{attribute 'qualified_only'}
{attribute 'strict'}
TYPE E_NoveltyDetectorType :
(
	KMPP := 0,
	KNN,
	LBG,
	NBC,
	STA,
	SVM
);
END_TYPE

(* stored: Version 1.1.0.1, ProductVersion 3.1.4024.12
   DUT E_NoveltyDetectorType: Id {b52dccab-d2ed-4c5e-9dae-8b721c3cc2ff} *)
